{attribute addProperty BoxType "KL2531-0001"}
{attribute addProperty Id "StatusAT %I*USINT000PositionAT %I*UDINT000ExtStatusAT %I*UINT000CtrlAT %Q*USINT000VelocityAT %Q*DINT000ExtCtrlAT %Q*UINT000"}
{attribute addProperty CRC "1429834296"}
{attribute addProperty SizeInBites "0"}
{attribute addProperty SizeInBytes "0"}
TYPE Channel_55398A38 :
STRUCT
	{attribute addProperty Name "Status"}
	Status AT %I* : USINT;
	{attribute addProperty Name "Position"}
	Position AT %I* : UDINT;
	{attribute addProperty Name "ExtStatus"}
	ExtStatus AT %I* : UINT;
	{attribute addProperty Name "Ctrl"}
	Ctrl AT %Q* : USINT;
	{attribute addProperty Name "Velocity"}
	Velocity AT %Q* : DINT;
	{attribute addProperty Name "ExtCtrl"}
	ExtCtrl AT %Q* : UINT;
END_STRUCT
END_TYPE

(* stored: Version 1.2.0.0, ProductVersion 3.1.4024.9
   DUT Channel_55398A38: Id {e33ed570-1c11-41e5-9b43-e54eef318fc2} *)
